{attribute 'qualified_only'}
{attribute 'strict'}
TYPE ENUM_UnitState :
(
  
	DISABLED := 1,
  OPERATIONAL :=2,
  STANDBY :=3,
  UNKNOWN :=4

);
END_TYPE

(* stored: Version 1.1.0.1, ProductVersion 3.1.4024.12
   DUT ENUM_UnitState: Id {8699ea60-09fc-4379-8ea8-50b536b47ef7} *)
